// NETWORK 2
fbStation2(in_strUniqueId := 'Station 2', in_fbDevice := fbDevice2); // FB_ExampleStation
END_ACTION

ACTION A_Station3:
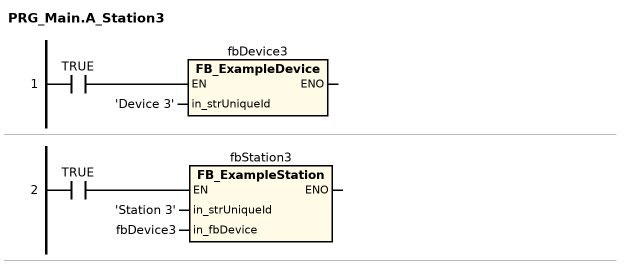
// NETWORK 1
fbDevice3(in_strUniqueId := 'Device 3'); // FB_ExampleDevice

// NETWORK 2
fbStation3(in_strUniqueId := 'Station 3', in_fbDevice := fbDevice3); // FB_ExampleStation
END_ACTION

ACTION A_Station4:
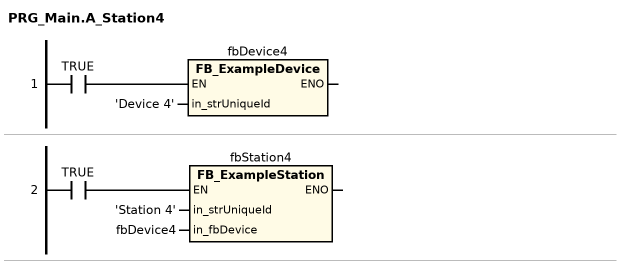
// NETWORK 1
fbDevice4(in_strUniqueId := 'Device 4'); // FB_ExampleDevice

// NETWORK 2
fbStation4(in_strUniqueId := 'Station 4', in_fbDevice := fbDevice4); // FB_ExampleStation
END_ACTION

METHOD M_TestCohapLibrary : BOOL

VAR
//	//Testing Cohap Related Vars

//	//Initialize Only	
//	MyCohapTest : FB_COHAP;
//	bInitializeCohapSystem: BOOL;
//	bRes_CohapConnected: BOOL;

//	//Execute RunImpMethods Only	;
//	bExecuteRunImpMethods: BOOL;
//	bRes_RunImpMethods: BOOL;

//	//Set Current Device Instance
//	bSetCurrentDevice_Cohap : BOOL;
//	bRes_SetCurrentDevice : BOOL;
//	//Input Params
//	strDeviceName : STRING;
	
//	//RunCommand
//	bRunCommandCohapSystem : BOOL;
//	bRes_RunCommand : BOOL;
//	//Input Params
//	strMethodName : STRING;
//	RunCom_InpuParams : T_CohapParameterList;
//	RunCom_ExpOutParamList : ARRAY[0..9] OF ST_ReturnParamsInfo;
//	//Output Params
//	RunCom_OutputParams : T_CohapParameterList;
	
//	//DummyTest Dictionary Prep for RunCommand Execution
//	RC_DT_InpPar : T_CohapParameterList;
//	RC_DT_ExpOutPL : ARRAY[0..9] OF ST_ReturnParamsInfo;
	
//	CohapMethodStrings : TMethodNames_Cohap;
//	CohapMethodControls : TMethod_Controls;
////	fbCohapHandler1: FB_COHAP;

/////////////////////////////////

//	// For readSerialNumber
//	readSerialNumber_inpuparams : T_CohapParameterList;
//	readSerialNumber_expoutparamlist : ARRAY[0..9] OF ST_ReturnParamsInfo;
//	readSerialNumber_outputparams : T_CohapParameterList;
	
//	// For ReadDeviceOutput
//	ReadDeviceOutput_inpuparams : T_CohapParameterList;
//	ReadDeviceOutput_expoutparamlist : ARRAY[0..9] OF ST_ReturnParamsInfo;
//	ReadDeviceOutput_outputparams : T_CohapParameterList;

	
//	// For PowerUp
//	PowerUp_inpuparams : T_CohapParameterList;
//	PowerUp_expoutparamlist : ARRAY[0..9] OF ST_ReturnParamsInfo;
//	PowerUp_outputparams : T_CohapParameterList;
	
//	// For PowerDown
//	PowerDown_inpuparams : T_CohapParameterList;
//	PowerDown_expoutparamlist : ARRAY[0..9] OF ST_ReturnParamsInfo;
//	PowerDown_outputparams : T_CohapParameterList;
	
//	// For TestDummy
//	TestDummy_inpuparams : T_CohapParameterList;
//	TestDummy_expoutparamlist : ARRAY[0..9] OF ST_ReturnParamsInfo;
//	TestDummy_outputparams : T_CohapParameterList;
	
//	// For TestDummy2
//	TestDummy2_inpuparams : T_CohapParameterList;
//	TestDummy2_expoutparamlist : ARRAY[0..9] OF ST_ReturnParamsInfo;
//	TestDummy2_outputparams : T_CohapParameterList;
	
//	// For init
//	init_inpuparams : T_CohapParameterList;
//	init_expoutparamlist : ARRAY[0..9] OF ST_ReturnParamsInfo;
//	init_outputparams : T_CohapParameterList;
	
//	// For getSICAndChannelCardVersions
//	getSICAndChannelCardVersions_inpuparams : T_CohapParameterList;
//	getSICAndChannelCardVersions_expoutparamlist : ARRAY[0..9] OF ST_ReturnParamsInfo;
//	getSICAndChannelCardVersions_outputparams : T_CohapParameterList;
	
//	// For getDLLVersions
//	getDLLVersions_inpuparams : T_CohapParameterList;
//	getDLLVersions_expoutparamlist : ARRAY[0..9] OF ST_ReturnParamsInfo;
//	getDLLVersions_outputparams : T_CohapParameterList;
	
//	// For initDUT
//	initDUT_inpuparams : T_CohapParameterList;
//	initDUT_expoutparamlist : ARRAY[0..9] OF ST_ReturnParamsInfo;
//	initDUT_outputparams : T_CohapParameterList;
	
//	//For Fast Channel Data
//	readFastChannelData_inputparams : T_CohapParameterList;
//	readFastChannelData_expoutparamlist : ARRAY[0..9] OF ST_ReturnParamsInfo;
//	readFastChannelData_outputparams : T_CohapParameterList;

//	// For T1 Step 1 Calibration
//	t1Step1_inpuparams : T_CohapParameterList;
//	t1Step1_expoutparamlist : ARRAY[0..9] OF ST_ReturnParamsInfo;
//	t1Step1_outputparams : T_CohapParameterList;
	
////	// For T1 Step 2 Calibration
////	t1Step2_inpuparams : T_CohapParameterList;
////	t1Step2_expoutparamlist : ARRAY[0..9] OF ST_ReturnParamsInfo;
////	t1Step2_outputparams : T_CohapParameterList;
	
////	// For T1 Step 3 Calibration
////	t1Step3_inpuparams : T_CohapParameterList;
////	t1Step3_expoutparamlist : ARRAY[0..9] OF ST_ReturnParamsInfo;
////	t1Step3_outputparams : T_CohapParameterList;
	
//	// For T2 Step 1 Calibration
//	t2Step1_inpuparams : T_CohapParameterList;
//	t2Step1_expoutparamlist : ARRAY[0..9] OF ST_ReturnParamsInfo;
//	t2Step1_outputparams : T_CohapParameterList;
	
//	// For T2 Step 2 Calibration
//	t2Step2_inpuparams : T_CohapParameterList;
//	t2Step2_expoutparamlist : ARRAY[0..9] OF ST_ReturnParamsInfo;
//	t2Step2_outputparams : T_CohapParameterList;
	
//	// For T2 Step 3 Calibration
//	t2Step3_inpuparams : T_CohapParameterList;
//	t2Step3_expoutparamlist : ARRAY[0..9] OF ST_ReturnParamsInfo;
//	t2Step3_outputparams : T_CohapParameterList;
	
//	// InitLot Device12133 class in Mech Device Lib Calibration
//	InitLot_inputparams : T_CohapParameterList;
//	InitLot_expoutparamlist : ARRAY[0..9] OF ST_ReturnParamsInfo;
//	InitLot_outputparams : T_CohapParameterList;
	
////	//For Init Lot
////	InitLot_inputparams : T_CohapParameterList;
////	InitLot_expoutparamlist : ARRAY[0..9] OF ST_ReturnParamsInfo;
////	InitLot_outputparams : T_CohapParameterList;	
//	// For T1 Step 1 Calibration
//	t1Precal_inputparams : T_CohapParameterList;
//	t1Precal_expoutparamlist : ARRAY[0..9] OF ST_ReturnParamsInfo;
//	t1Precal_outputparams : T_CohapParameterList;
//	// For T1 Step 2 Calibration
//	t1Step2_inputparams : T_CohapParameterList;
//	t1Step2_expoutparamlist : ARRAY[0..9] OF ST_ReturnParamsInfo;
//	t1Step2_outputparams : T_CohapParameterList;
//	// For T1 Step 3 Calibration
//	t1Step3_inputparams : T_CohapParameterList;
//	t1Step3_expoutparamlist : ARRAY[0..9] OF ST_ReturnParamsInfo;
//	t1Step3_outputparams : T_CohapParameterList;
END_VAR
VAR_INST // added by the converter: edge detectors and wires of the graphical bodies
    _w1, _w2, _w3, _w4, _w5, _w6, _w7, _w8, _w9, _w10, _w11, _w12, _w13, _w14, _w15, _w16, _w17, _w18, _w19, _w20, _w21, _w22, _w23, _w24, _w25, _w26, _w27, _w28, _w29, _w30, _w31, _w32, _w33, _w34, _w35, _w36, _w37, _w38, _w39, _w40 : BOOL;
END_VAR
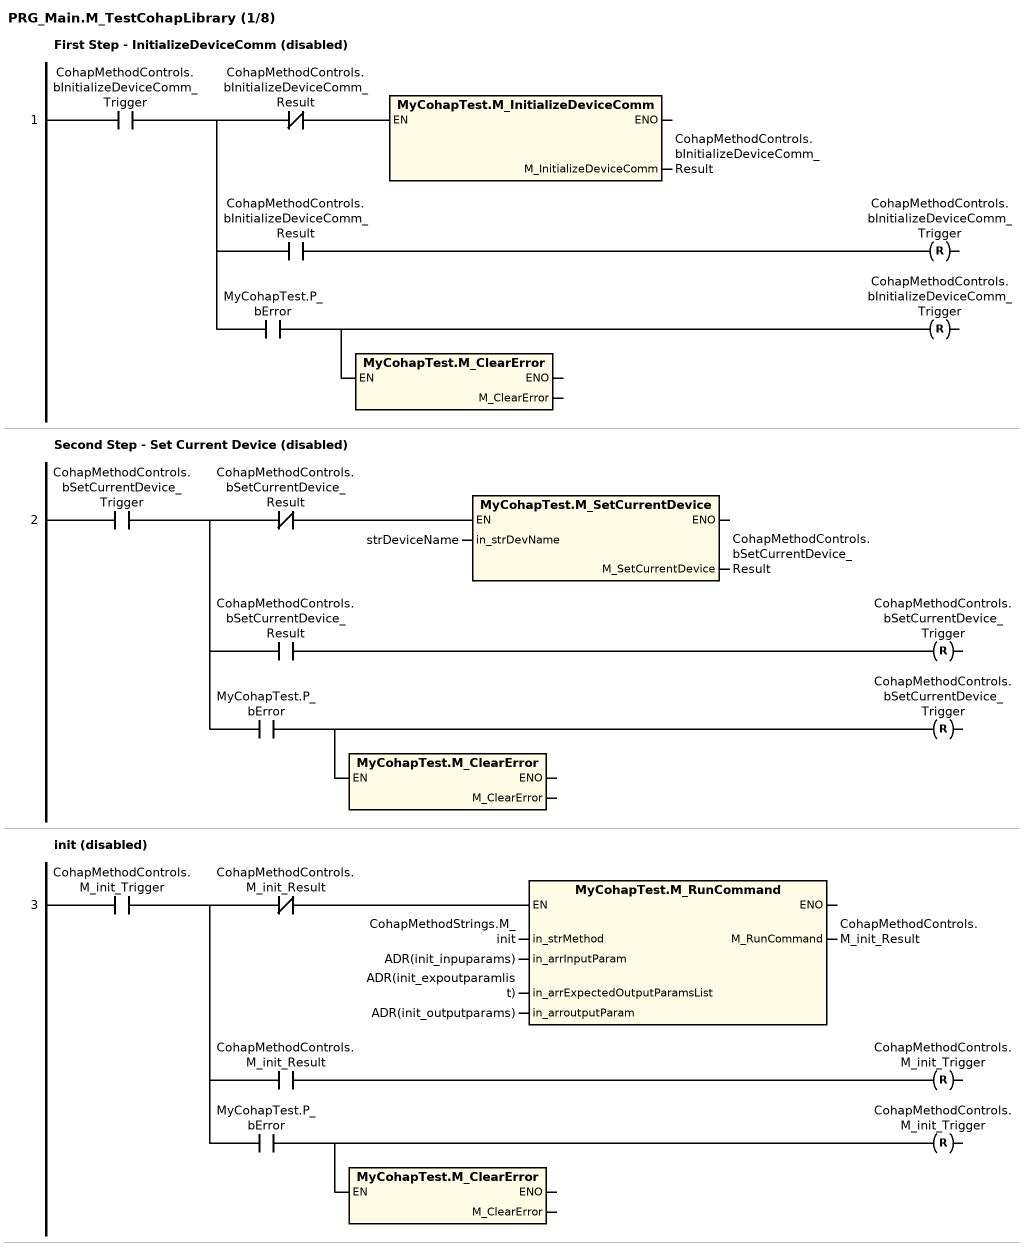
// NETWORK 1: First Step - InitializeDeviceComm (disabled)
// _w1 := CohapMethodControls.bInitializeDeviceComm_Trigger;
// IF _w1 AND NOT CohapMethodControls.bInitializeDeviceComm_Result THEN
//     CohapMethodControls.bInitializeDeviceComm_Result := MyCohapTest.M_InitializeDeviceComm();
// END_IF
// CohapMethodControls.bInitializeDeviceComm_Trigger R= _w1 AND CohapMethodControls.bInitializeDeviceComm_Result;
// _w2 := _w1 AND MyCohapTest.P_bError;
// CohapMethodControls.bInitializeDeviceComm_Trigger R= _w2;
// IF _w2 THEN MyCohapTest.M_ClearError(); END_IF

// NETWORK 2: Second Step - Set Current Device (disabled)
// _w3 := CohapMethodControls.bSetCurrentDevice_Trigger;
// IF _w3 AND NOT CohapMethodControls.bSetCurrentDevice_Result THEN
//     CohapMethodControls.bSetCurrentDevice_Result := MyCohapTest.M_SetCurrentDevice(in_strDevName := strDeviceName);
// END_IF
// CohapMethodControls.bSetCurrentDevice_Trigger R= _w3 AND CohapMethodControls.bSetCurrentDevice_Result;
// _w4 := _w3 AND MyCohapTest.P_bError;
// CohapMethodControls.bSetCurrentDevice_Trigger R= _w4;
// IF _w4 THEN MyCohapTest.M_ClearError(); END_IF

// NETWORK 3: init (disabled)
// _w5 := CohapMethodControls.M_init_Trigger;
// IF _w5 AND NOT CohapMethodControls.M_init_Result THEN
//     CohapMethodControls.M_init_Result := MyCohapTest.M_RunCommand(in_strMethod := CohapMethodStrings.M_init, in_arrInputParam := ADR(init_inpuparams), in_arrExpectedOutputParamsList := ADR(init_expoutparamlist), in_arroutputParam := ADR(init_outputparams));
// END_IF
// CohapMethodControls.M_init_Trigger R= _w5 AND CohapMethodControls.M_init_Result;
// _w6 := _w5 AND MyCohapTest.P_bError;
// CohapMethodControls.M_init_Trigger R= _w6;
// IF _w6 THEN MyCohapTest.M_ClearError(); END_IF

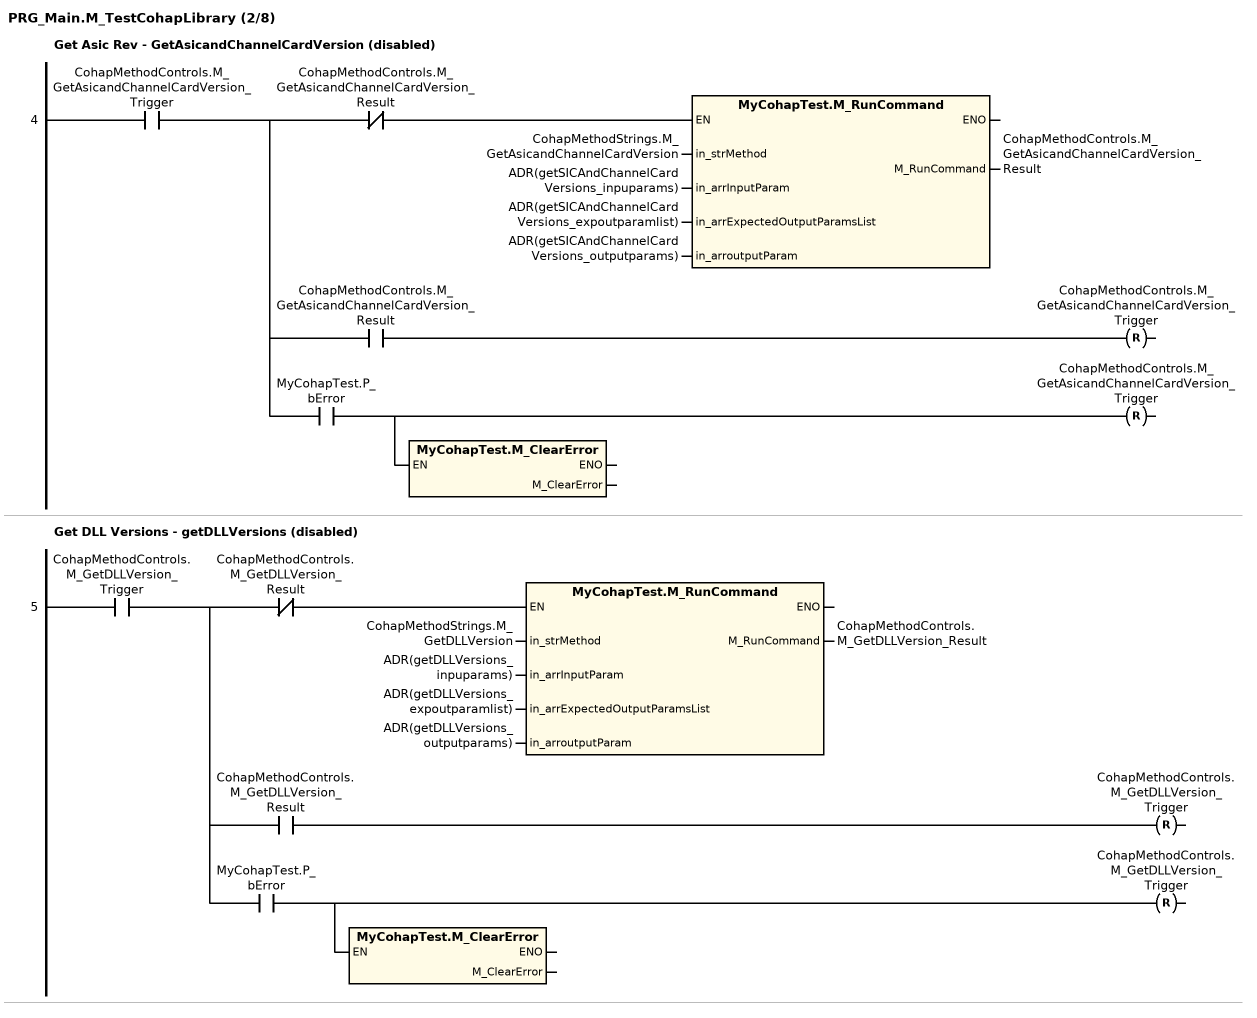
// NETWORK 4: Get Asic Rev - GetAsicandChannelCardVersion (disabled)
// _w7 := CohapMethodControls.M_GetAsicandChannelCardVersion_Trigger;
// IF _w7 AND NOT CohapMethodControls.M_GetAsicandChannelCardVersion_Result THEN
//     CohapMethodControls.M_GetAsicandChannelCardVersion_Result := MyCohapTest.M_RunCommand(in_strMethod := CohapMethodStrings.M_GetAsicandChannelCardVersion, in_arrInputParam := ADR(getSICAndChannelCardVersions_inpuparams), in_arrExpectedOutputParamsList := ADR(getSICAndChannelCardVersions_expoutparamlist), in_arroutputParam := ADR(getSICAndChannelCardVersions_outputparams));
// END_IF
// CohapMethodControls.M_GetAsicandChannelCardVersion_Trigger R= _w7 AND CohapMethodControls.M_GetAsicandChannelCardVersion_Result;
// _w8 := _w7 AND MyCohapTest.P_bError;
// CohapMethodControls.M_GetAsicandChannelCardVersion_Trigger R= _w8;
// IF _w8 THEN MyCohapTest.M_ClearError(); END_IF

// NETWORK 5: Get DLL Versions - getDLLVersions (disabled)
// _w9 := CohapMethodControls.M_GetDLLVersion_Trigger;
// IF _w9 AND NOT CohapMethodControls.M_GetDLLVersion_Result THEN
//     CohapMethodControls.M_GetDLLVersion_Result := MyCohapTest.M_RunCommand(in_strMethod := CohapMethodStrings.M_GetDLLVersion, in_arrInputParam := ADR(getDLLVersions_inpuparams), in_arrExpectedOutputParamsList := ADR(getDLLVersions_expoutparamlist), in_arroutputParam := ADR(getDLLVersions_outputparams));
// END_IF
// CohapMethodControls.M_GetDLLVersion_Trigger R= _w9 AND CohapMethodControls.M_GetDLLVersion_Result;
// _w10 := _w9 AND MyCohapTest.P_bError;
// CohapMethodControls.M_GetDLLVersion_Trigger R= _w10;
// IF _w10 THEN MyCohapTest.M_ClearError(); END_IF

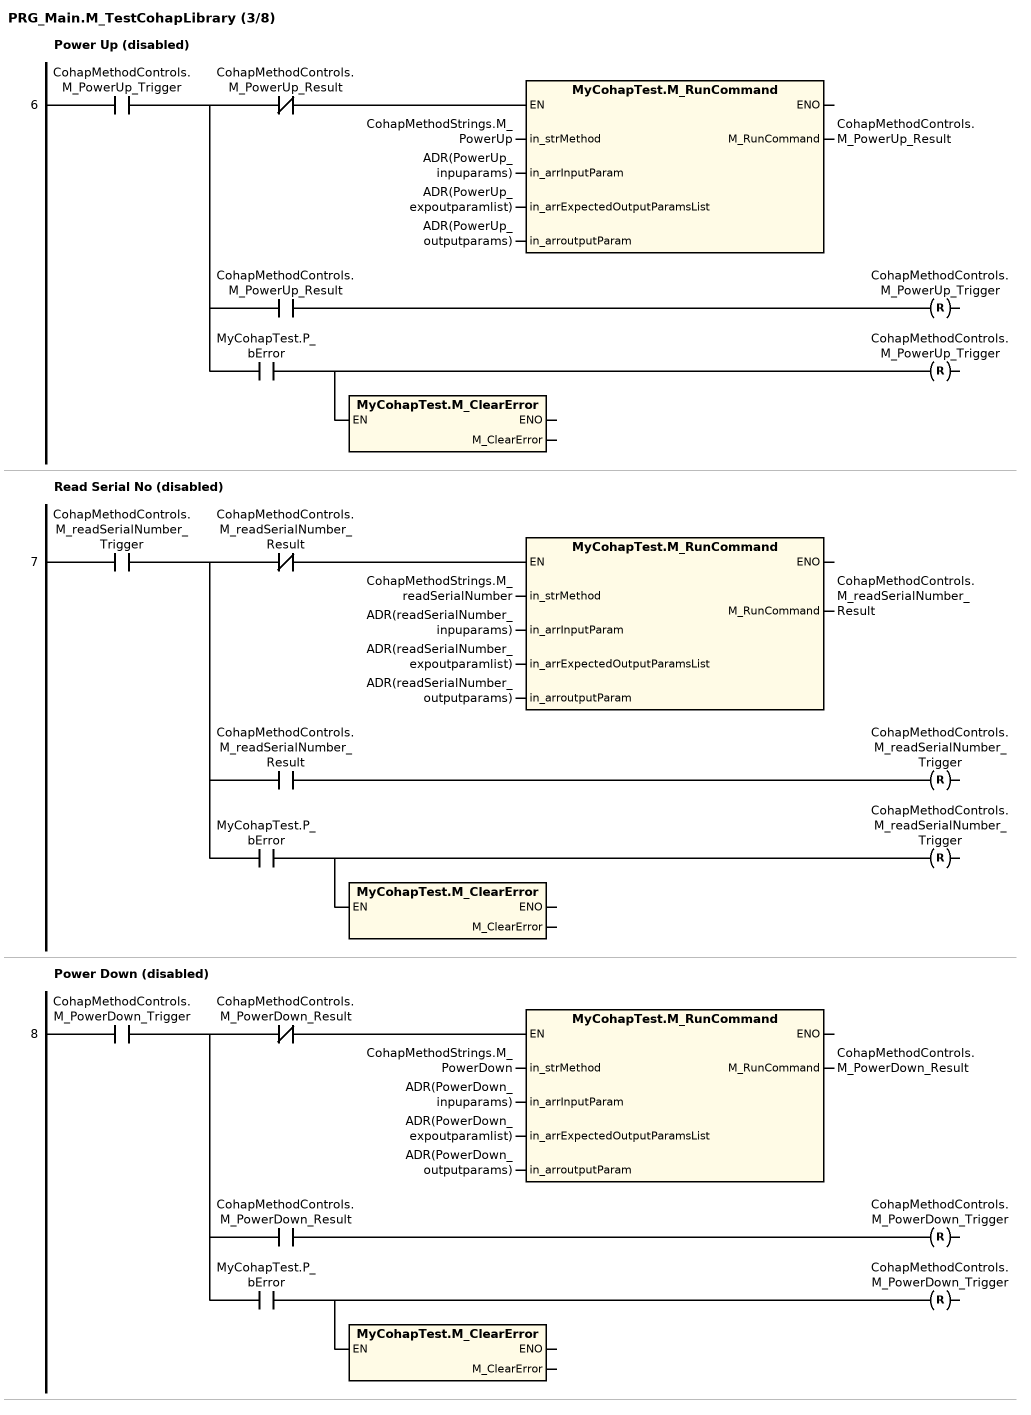
// NETWORK 6: Power Up (disabled)
// _w11 := CohapMethodControls.M_PowerUp_Trigger;
// IF _w11 AND NOT CohapMethodControls.M_PowerUp_Result THEN
//     CohapMethodControls.M_PowerUp_Result := MyCohapTest.M_RunCommand(in_strMethod := CohapMethodStrings.M_PowerUp, in_arrInputParam := ADR(PowerUp_inpuparams), in_arrExpectedOutputParamsList := ADR(PowerUp_expoutparamlist), in_arroutputParam := ADR(PowerUp_outputparams));
// END_IF
// CohapMethodControls.M_PowerUp_Trigger R= _w11 AND CohapMethodControls.M_PowerUp_Result;
// _w12 := _w11 AND MyCohapTest.P_bError;
// CohapMethodControls.M_PowerUp_Trigger R= _w12;
// IF _w12 THEN MyCohapTest.M_ClearError(); END_IF

// NETWORK 7: Read Serial No (disabled)
// _w13 := CohapMethodControls.M_readSerialNumber_Trigger;
// IF _w13 AND NOT CohapMethodControls.M_readSerialNumber_Result THEN
//     CohapMethodControls.M_readSerialNumber_Result := MyCohapTest.M_RunCommand(in_strMethod := CohapMethodStrings.M_readSerialNumber, in_arrInputParam := ADR(readSerialNumber_inpuparams), in_arrExpectedOutputParamsList := ADR(readSerialNumber_expoutparamlist), in_arroutputParam := ADR(readSerialNumber_outputparams));
// END_IF
// CohapMethodControls.M_readSerialNumber_Trigger R= _w13 AND CohapMethodControls.M_readSerialNumber_Result;
// _w14 := _w13 AND MyCohapTest.P_bError;
// CohapMethodControls.M_readSerialNumber_Trigger R= _w14;
// IF _w14 THEN MyCohapTest.M_ClearError(); END_IF

// NETWORK 8: Power Down (disabled)
// _w15 := CohapMethodControls.M_PowerDown_Trigger;
// IF _w15 AND NOT CohapMethodControls.M_PowerDown_Result THEN
//     CohapMethodControls.M_PowerDown_Result := MyCohapTest.M_RunCommand(in_strMethod := CohapMethodStrings.M_PowerDown, in_arrInputParam := ADR(PowerDown_inpuparams), in_arrExpectedOutputParamsList := ADR(PowerDown_expoutparamlist), in_arroutputParam := ADR(PowerDown_outputparams));
// END_IF
// CohapMethodControls.M_PowerDown_Trigger R= _w15 AND CohapMethodControls.M_PowerDown_Result;
// _w16 := _w15 AND MyCohapTest.P_bError;
// CohapMethodControls.M_PowerDown_Trigger R= _w16;
// IF _w16 THEN MyCohapTest.M_ClearError(); END_IF

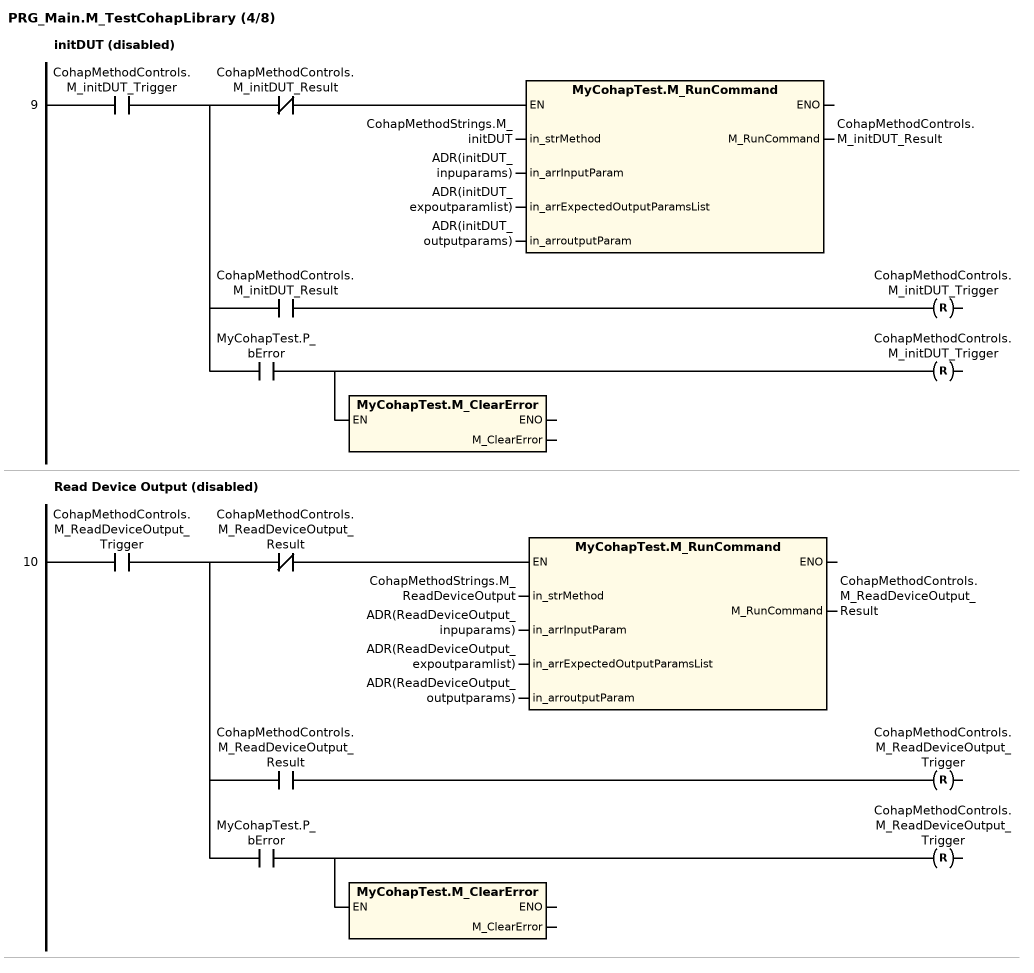
// NETWORK 9: initDUT (disabled)
// _w17 := CohapMethodControls.M_initDUT_Trigger;
// IF _w17 AND NOT CohapMethodControls.M_initDUT_Result THEN
//     CohapMethodControls.M_initDUT_Result := MyCohapTest.M_RunCommand(in_strMethod := CohapMethodStrings.M_initDUT, in_arrInputParam := ADR(initDUT_inpuparams), in_arrExpectedOutputParamsList := ADR(initDUT_expoutparamlist), in_arroutputParam := ADR(initDUT_outputparams));
// END_IF
// CohapMethodControls.M_initDUT_Trigger R= _w17 AND CohapMethodControls.M_initDUT_Result;
// _w18 := _w17 AND MyCohapTest.P_bError;
// CohapMethodControls.M_initDUT_Trigger R= _w18;
// IF _w18 THEN MyCohapTest.M_ClearError(); END_IF

// NETWORK 10: Read Device Output (disabled)
// _w19 := CohapMethodControls.M_ReadDeviceOutput_Trigger;
// IF _w19 AND NOT CohapMethodControls.M_ReadDeviceOutput_Result THEN
//     CohapMethodControls.M_ReadDeviceOutput_Result := MyCohapTest.M_RunCommand(in_strMethod := CohapMethodStrings.M_ReadDeviceOutput, in_arrInputParam := ADR(ReadDeviceOutput_inpuparams), in_arrExpectedOutputParamsList := ADR(ReadDeviceOutput_expoutparamlist), in_arroutputParam := ADR(ReadDeviceOutput_outputparams));
// END_IF
// CohapMethodControls.M_ReadDeviceOutput_Trigger R= _w19 AND CohapMethodControls.M_ReadDeviceOutput_Result;
// _w20 := _w19 AND MyCohapTest.P_bError;
// CohapMethodControls.M_ReadDeviceOutput_Trigger R= _w20;
// IF _w20 THEN MyCohapTest.M_ClearError(); END_IF

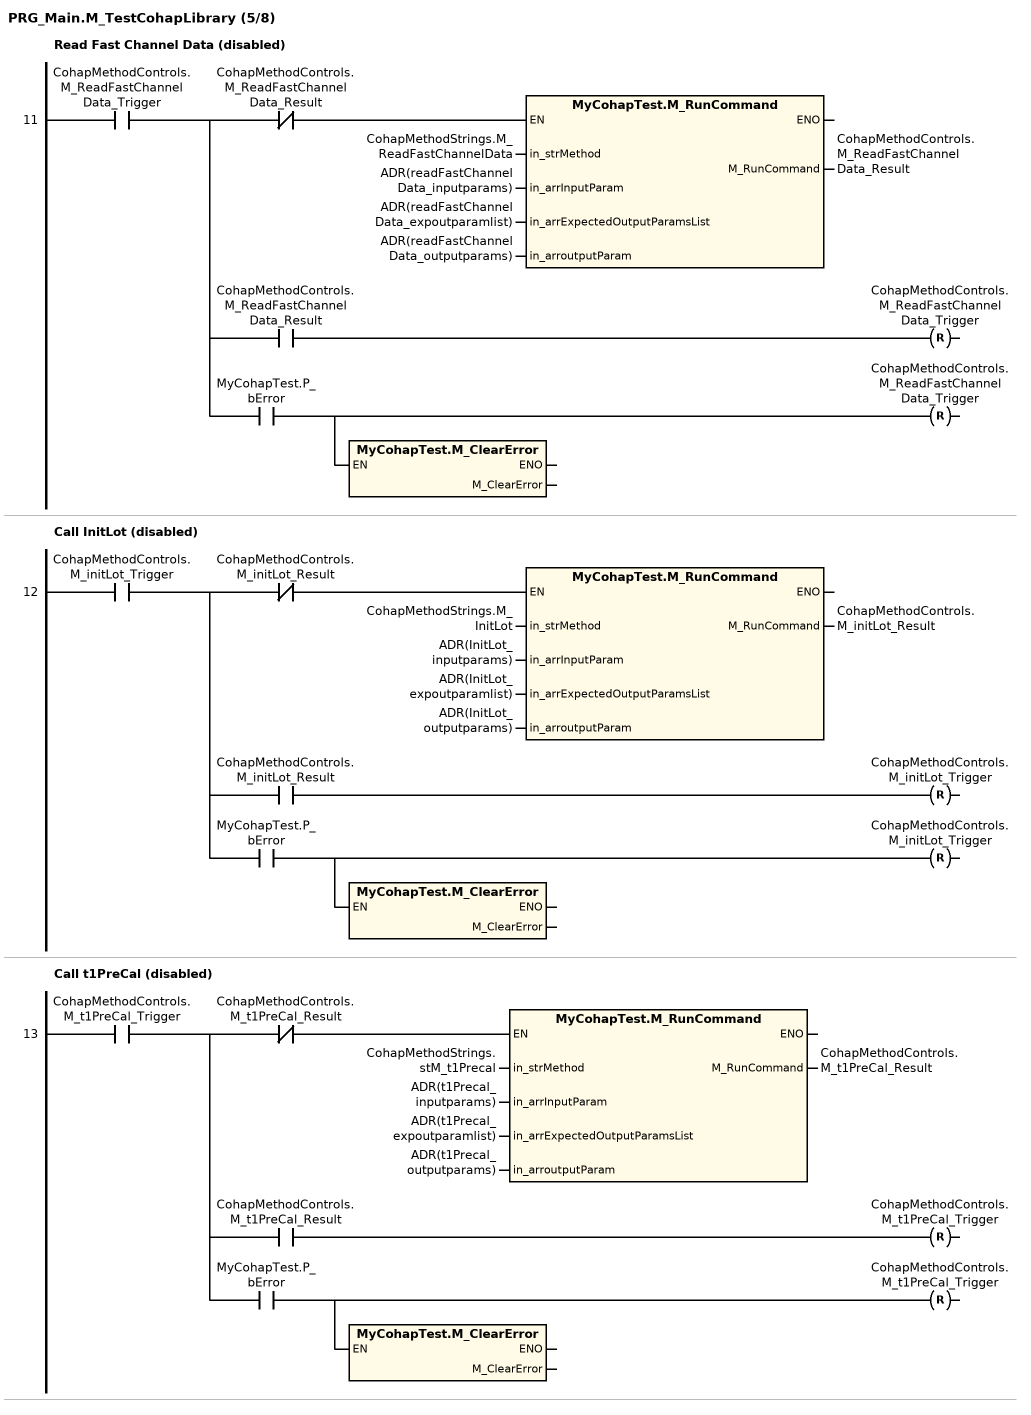
// NETWORK 11: Read Fast Channel Data (disabled)
// _w21 := CohapMethodControls.M_ReadFastChannelData_Trigger;
// IF _w21 AND NOT CohapMethodControls.M_ReadFastChannelData_Result THEN
//     CohapMethodControls.M_ReadFastChannelData_Result := MyCohapTest.M_RunCommand(in_strMethod := CohapMethodStrings.M_ReadFastChannelData, in_arrInputParam := ADR(readFastChannelData_inputparams), in_arrExpectedOutputParamsList := ADR(readFastChannelData_expoutparamlist), in_arroutputParam := ADR(readFastChannelData_outputparams));
// END_IF
// CohapMethodControls.M_ReadFastChannelData_Trigger R= _w21 AND CohapMethodControls.M_ReadFastChannelData_Result;
// _w22 := _w21 AND MyCohapTest.P_bError;
// CohapMethodControls.M_ReadFastChannelData_Trigger R= _w22;
// IF _w22 THEN MyCohapTest.M_ClearError(); END_IF

// NETWORK 12: Call InitLot (disabled)
// _w23 := CohapMethodControls.M_initLot_Trigger;
// IF _w23 AND NOT CohapMethodControls.M_initLot_Result THEN
//     CohapMethodControls.M_initLot_Result := MyCohapTest.M_RunCommand(in_strMethod := CohapMethodStrings.M_InitLot, in_arrInputParam := ADR(InitLot_inputparams), in_arrExpectedOutputParamsList := ADR(InitLot_expoutparamlist), in_arroutputParam := ADR(InitLot_outputparams));
// END_IF
// CohapMethodControls.M_initLot_Trigger R= _w23 AND CohapMethodControls.M_initLot_Result;
// _w24 := _w23 AND MyCohapTest.P_bError;
// CohapMethodControls.M_initLot_Trigger R= _w24;
// IF _w24 THEN MyCohapTest.M_ClearError(); END_IF

// NETWORK 13: Call t1PreCal (disabled)
// _w25 := CohapMethodControls.M_t1PreCal_Trigger;
// IF _w25 AND NOT CohapMethodControls.M_t1PreCal_Result THEN
//     CohapMethodControls.M_t1PreCal_Result := MyCohapTest.M_RunCommand(in_strMethod := CohapMethodStrings.stM_t1Precal, in_arrInputParam := ADR(t1Precal_inputparams), in_arrExpectedOutputParamsList := ADR(t1Precal_expoutparamlist), in_arroutputParam := ADR(t1Precal_outputparams));
// END_IF
// CohapMethodControls.M_t1PreCal_Trigger R= _w25 AND CohapMethodControls.M_t1PreCal_Result;
// _w26 := _w25 AND MyCohapTest.P_bError;
// CohapMethodControls.M_t1PreCal_Trigger R= _w26;
// IF _w26 THEN MyCohapTest.M_ClearError(); END_IF

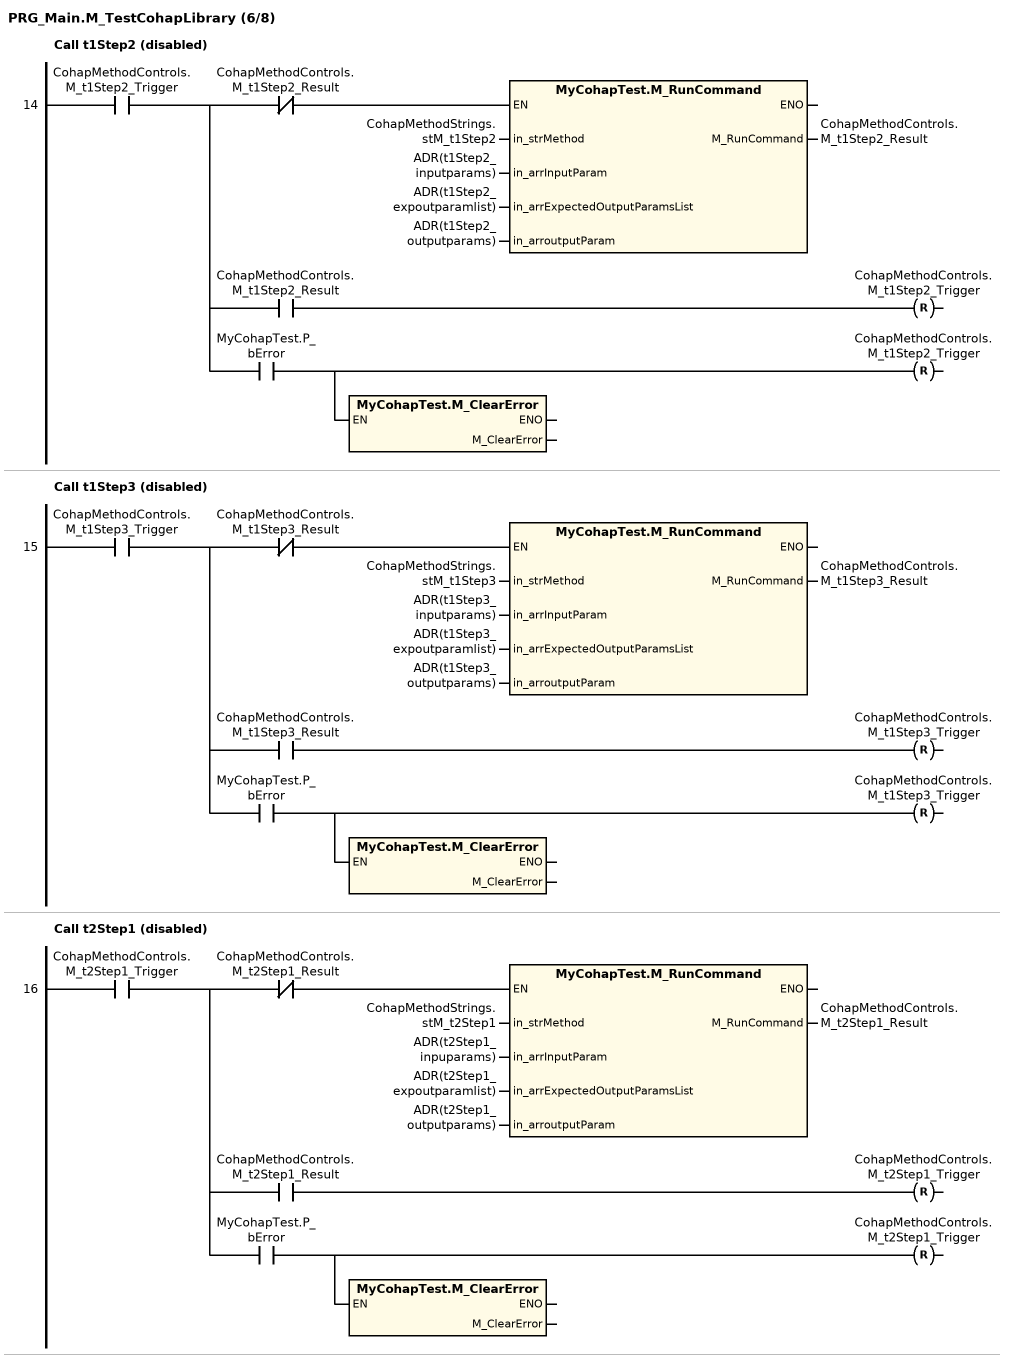
// NETWORK 14: Call t1Step2 (disabled)
// _w27 := CohapMethodControls.M_t1Step2_Trigger;
// IF _w27 AND NOT CohapMethodControls.M_t1Step2_Result THEN
//     CohapMethodControls.M_t1Step2_Result := MyCohapTest.M_RunCommand(in_strMethod := CohapMethodStrings.stM_t1Step2, in_arrInputParam := ADR(t1Step2_inputparams), in_arrExpectedOutputParamsList := ADR(t1Step2_expoutparamlist), in_arroutputParam := ADR(t1Step2_outputparams));
// END_IF
// CohapMethodControls.M_t1Step2_Trigger R= _w27 AND CohapMethodControls.M_t1Step2_Result;
// _w28 := _w27 AND MyCohapTest.P_bError;
// CohapMethodControls.M_t1Step2_Trigger R= _w28;
// IF _w28 THEN MyCohapTest.M_ClearError(); END_IF

// NETWORK 15: Call t1Step3 (disabled)
// _w29 := CohapMethodControls.M_t1Step3_Trigger;
// IF _w29 AND NOT CohapMethodControls.M_t1Step3_Result THEN
//     CohapMethodControls.M_t1Step3_Result := MyCohapTest.M_RunCommand(in_strMethod := CohapMethodStrings.stM_t1Step3, in_arrInputParam := ADR(t1Step3_inputparams), in_arrExpectedOutputParamsList := ADR(t1Step3_expoutparamlist), in_arroutputParam := ADR(t1Step3_outputparams));
// END_IF
// CohapMethodControls.M_t1Step3_Trigger R= _w29 AND CohapMethodControls.M_t1Step3_Result;
// _w30 := _w29 AND MyCohapTest.P_bError;
// CohapMethodControls.M_t1Step3_Trigger R= _w30;
// IF _w30 THEN MyCohapTest.M_ClearError(); END_IF

// NETWORK 16: Call t2Step1 (disabled)
// _w31 := CohapMethodControls.M_t2Step1_Trigger;
// IF _w31 AND NOT CohapMethodControls.M_t2Step1_Result THEN
//     CohapMethodControls.M_t2Step1_Result := MyCohapTest.M_RunCommand(in_strMethod := CohapMethodStrings.stM_t2Step1, in_arrInputParam := ADR(t2Step1_inpuparams), in_arrExpectedOutputParamsList := ADR(t2Step1_expoutparamlist), in_arroutputParam := ADR(t2Step1_outputparams));
// END_IF
// CohapMethodControls.M_t2Step1_Trigger R= _w31 AND CohapMethodControls.M_t2Step1_Result;
// _w32 := _w31 AND MyCohapTest.P_bError;
// CohapMethodControls.M_t2Step1_Trigger R= _w32;
// IF _w32 THEN MyCohapTest.M_ClearError(); END_IF

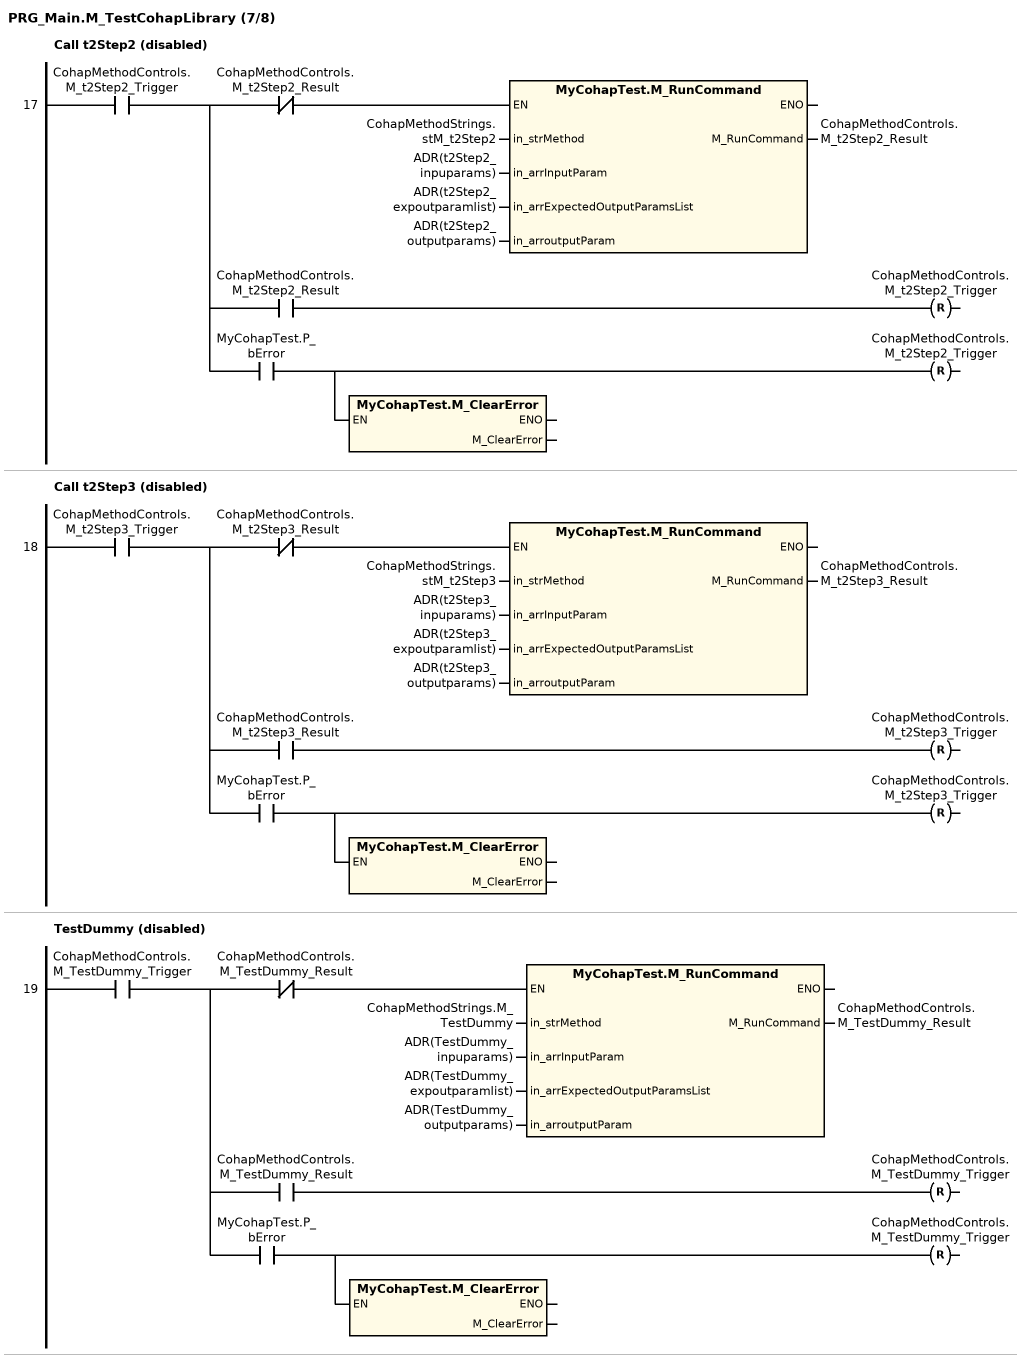
// NETWORK 17: Call t2Step2 (disabled)
// _w33 := CohapMethodControls.M_t2Step2_Trigger;
// IF _w33 AND NOT CohapMethodControls.M_t2Step2_Result THEN
//     CohapMethodControls.M_t2Step2_Result := MyCohapTest.M_RunCommand(in_strMethod := CohapMethodStrings.stM_t2Step2, in_arrInputParam := ADR(t2Step2_inpuparams), in_arrExpectedOutputParamsList := ADR(t2Step2_expoutparamlist), in_arroutputParam := ADR(t2Step2_outputparams));
// END_IF
// CohapMethodControls.M_t2Step2_Trigger R= _w33 AND CohapMethodControls.M_t2Step2_Result;
// _w34 := _w33 AND MyCohapTest.P_bError;
// CohapMethodControls.M_t2Step2_Trigger R= _w34;
// IF _w34 THEN MyCohapTest.M_ClearError(); END_IF

// NETWORK 18: Call t2Step3 (disabled)
// _w35 := CohapMethodControls.M_t2Step3_Trigger;
// IF _w35 AND NOT CohapMethodControls.M_t2Step3_Result THEN
//     CohapMethodControls.M_t2Step3_Result := MyCohapTest.M_RunCommand(in_strMethod := CohapMethodStrings.stM_t2Step3, in_arrInputParam := ADR(t2Step3_inpuparams), in_arrExpectedOutputParamsList := ADR(t2Step3_expoutparamlist), in_arroutputParam := ADR(t2Step3_outputparams));
// END_IF
// CohapMethodControls.M_t2Step3_Trigger R= _w35 AND CohapMethodControls.M_t2Step3_Result;
// _w36 := _w35 AND MyCohapTest.P_bError;
// CohapMethodControls.M_t2Step3_Trigger R= _w36;
// IF _w36 THEN MyCohapTest.M_ClearError(); END_IF

// NETWORK 19: TestDummy (disabled)
// _w37 := CohapMethodControls.M_TestDummy_Trigger;
// IF _w37 AND NOT CohapMethodControls.M_TestDummy_Result THEN
//     CohapMethodControls.M_TestDummy_Result := MyCohapTest.M_RunCommand(in_strMethod := CohapMethodStrings.M_TestDummy, in_arrInputParam := ADR(TestDummy_inpuparams), in_arrExpectedOutputParamsList := ADR(TestDummy_expoutparamlist), in_arroutputParam := ADR(TestDummy_outputparams));
// END_IF
// CohapMethodControls.M_TestDummy_Trigger R= _w37 AND CohapMethodControls.M_TestDummy_Result;
// _w38 := _w37 AND MyCohapTest.P_bError;
// CohapMethodControls.M_TestDummy_Trigger R= _w38;
// IF _w38 THEN MyCohapTest.M_ClearError(); END_IF

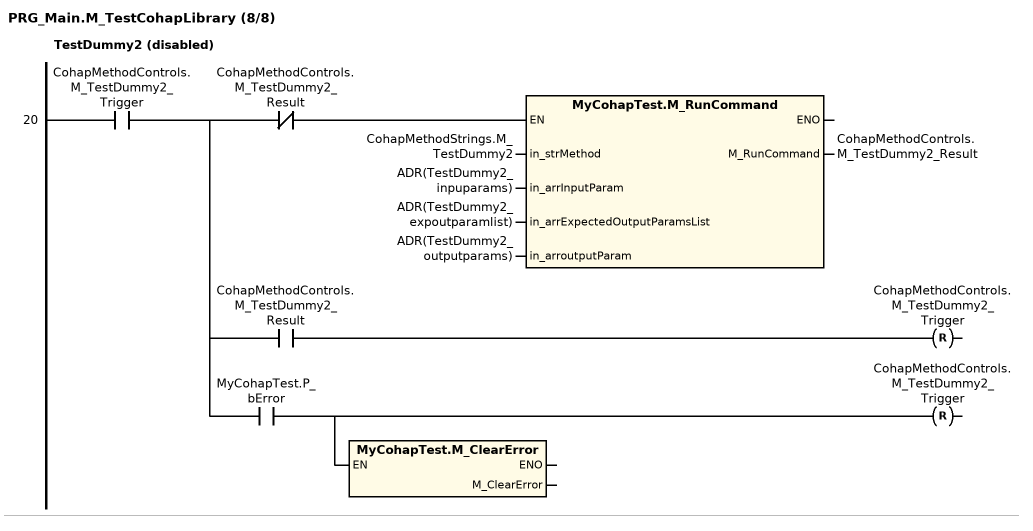
// NETWORK 20: TestDummy2 (disabled)
// _w39 := CohapMethodControls.M_TestDummy2_Trigger;
// IF _w39 AND NOT CohapMethodControls.M_TestDummy2_Result THEN
//     CohapMethodControls.M_TestDummy2_Result := MyCohapTest.M_RunCommand(in_strMethod := CohapMethodStrings.M_TestDummy2, in_arrInputParam := ADR(TestDummy2_inpuparams), in_arrExpectedOutputParamsList := ADR(TestDummy2_expoutparamlist), in_arroutputParam := ADR(TestDummy2_outputparams));
// END_IF
// CohapMethodControls.M_TestDummy2_Trigger R= _w39 AND CohapMethodControls.M_TestDummy2_Result;
// _w40 := _w39 AND MyCohapTest.P_bError;
// CohapMethodControls.M_TestDummy2_Trigger R= _w40;
// IF _w40 THEN MyCohapTest.M_ClearError(); END_IF
END_METHOD

METHOD M_TestLaserMarker : BOOL
VAR_INPUT
END_VAR
VAR
		bConnectToLaserMarker: BOOL;
	bRes_LaserConnected: BOOL;
	bTestADSServer: BOOL;
	strTarget: T_MaxString;
	strCommand: T_MaxString;
	arrParams: T_ApiMethodParameters;
	MyResults: T_MaxString;
	bInterfaceTest : BOOL;
	temp: BOOL;
	bDisconnectFromLaserMarker: BOOL;
	bRes_LaserDisconnected: BOOL;
	bPeakCurrentProgramInLaser: BOOL;
	bRes_PeakCurrentProgramInLaser: BOOL;
	bSendProgramToLaser: BOOL;
	bRes_SendProgramtoLaser: BOOL;
	filepath : STRING;
	LaserMemoryLocation : INT;
	bSaveCurrentLaserProgramtoPC : BOOL;
	bRes_SaveCurrentLaserProgramtoPC: BOOL;
	LaserProgramFolderPath: STRING;
	bGetCurrentProgram : BOOL;
	bRes_GetCurrentProgram : BOOL;
	CurrentProgramName : T_MaxString;
	bStartMarking: BOOL;
	bRes_StartMarking: BOOL;
	bStopMarking: BOOL;
	bRes_StopMarking: BOOL;
	bClearLaserErrors: BOOL;
	bRes_ClearLaserErrors: BOOL;
	bUpdateProgramBlockInTheLaser: BOOL;
	bRes_UpdateProgramBlockInTheLaser: BOOL;
	_blockNumber: INT;
	_blockData: STRING;
	_blockType : BlockTypes;
	bGetLaserStatus: BOOL;
	bRes_GetLaserStatus: BOOL;
	_string_laserstatus : STRING;
	bGetLaserErrorStatus: BOOL;
	bRes_GetLaserErrorStatus: BOOL;
	_bIsLaserError : BOOL;
	bGetLaserActivatedStatus: BOOL;
	bRes_GetLaserActivatedStatus: BOOL;
	_bIsLaserActivated : BOOL;
	bGetLaserMarkingStatus: BOOL;
	bRes_GetLaserMarkingStatus: BOOL;
	_bIsLaserMarking : BOOL;
	bRes_Reset: BOOL;
	bResetErrors: BOOL;
	bUpdateProgramBlockMarkEnabledInTheLaser: BOOL;
	bRes_UpdateProgramBlockMarkEnabledInTheLaser: BOOL;
	_bool_markenabled : BOOL;
	_blockType_enum : BlockTypes;
	UpdateSingleBlockMarkEnabledIntheLaser_Success: BOOL;
	_bUpdateSingleBlockDataSuccess : BOOL;
	_bUpdateSingleBlockMarkEnabled_Success : BOOL;
	bUpdateAllMarkingInfo: BOOL;
	LastBlockToMark : INT;
	_OneTimeArrayBuild : BOOL := TRUE;
	BlockInfoArray : ARRAY [0..255] OF OneBlockInfo;
	bRes_UpdateAllMarkingInfo: BOOL;
	intIndex: INT;
	intIndex2 : INT;
	inst_intStep: INT := 0;
	_tempString : STRING;
	bRes_UpdateAllMarkInfo : ARRAY [0..255] OF BOOL;
	bUpdateAllMarkingInfo_MethodCall: BOOL;
	bRes_UpdateAllMarkingInfo_MethodCall: BOOL;
	fbDataHandler: FB_DataTracker;
	fbDataHandler2: FB_DataTracker;
	fbDatabaseCommandRouter: FB_AdsCommandRouter;
	_inst_bDataTransferred: BOOL;
	// (* Name of the parameters database transfer ID. *)
	in_strParametersDatabaseName: T_MaxString := 'GetLimits';
	in_strParametersDBNameLaserLimits_L1 : T_MaxString := 'GetLaserMarkingParams_L1';
	in_strParametersDBNameLaserLimits_L2 : T_MaxString := 'GetLaserMarkingParams_L2';
	in_strParametersDBNameLaserLimits_R1 : T_MaxString := 'GetLaserMarkingParams_R1';
	in_strParametersDBNameLaserLimits_R2 : T_MaxString := 'GetLaserMarkingParams_R2';	
	_inst_bLaserLimitsDataTransferred_L1 : BOOL;
	_inst_bLaserLimitsDataTransferred_L2 : BOOL;
	_inst_bLaserLimitsDataTransferred_R1 : BOOL;
	_inst_bLaserLimitsDataTransferred_R2 : BOOL;
	bGetLimitsFromDB : BOOL;
	bGetLaserParamsFromDB_L1 : BOOL;
	bGetLaserParamsFromDB_L2 : BOOL;
	bGetLaserParamsFromDB_R1 : BOOL;
	bGetLaserParamsFromDB_R2 : BOOL;
	bPerformPriorOp_Smart: BOOL;
	in_strParametersDBName_SmartWater : T_MaxString := 'GetPriorOPA';
	_inst_bPriorOp_Smart: BOOL;
	
	bPerformPriorOp_FFT: BOOL;
	in_strParametersDBName_FFTLaser_L1 : T_MaxString := 'LaserMarkCheckL1';
	_inst_bPriorOp_FFT: BOOL;
	
	Temp_CR_LOOKUP_NestL1 : INT;
	iLengthDataMatrixNestL1 : INT;
	ParamsArrayNestA : STRING;
END_VAR
//IF bConnectToLaserMarker THEN
//	bRes_LaserConnected := MyLaser1.M_Connect();
//	IF bRes_LaserConnected THEN
//	//Add some timer based logic to do error handling.
//		bConnectToLaserMarker := FALSE;
//	ELSIF MyLaser1.P_bError THEN
//		bConnectToLaserMarker := FALSE;
//		MyLaser1.M_ClearError();
//	END_IF
//END_IF


//IF bDisconnectFromLaserMarker THEN
//	bRes_LaserDisconnected := MyLaser1.M_Disconnect();
//	IF bRes_LaserDisconnected THEN
//		bDisconnectFromLaserMarker := FALSE;
//	ELSIF MyLaser1.P_bError THEN
//		bDisconnectFromLaserMarker := FALSE;
//		MyLaser1.M_ClearError();
//	END_IF
//END_IF


//IF bPeakCurrentProgramInLaser THEN
//	bRes_PeakCurrentProgramInLaser := MyLaser1.M_PeakCurrentProgram();
//	IF bRes_PeakCurrentProgramInLaser THEN
//		bPeakCurrentProgramInLaser := FALSE;
//	ELSIF MyLaser1.P_bError THEN
//		bPeakCurrentProgramInLaser := FALSE;
//		MyLaser1.M_ClearError();
//	END_IF
//END_IF


//IF bSendProgramToLaser THEN
//	bRes_SendProgramtoLaser := MyLaser1.M_SendProgramtoLaser(filepath,LaserMemoryLocation);
//	IF bRes_SendProgramtoLaser THEN
//		bSendProgramToLaser := FALSE;
//	ELSIF MyLaser1.P_bError THEN
//		bSendProgramToLaser := FALSE;
//		MyLaser1.M_ClearError();
//	END_IF
//END_IF

//IF bSaveCurrentLaserProgramtoPC THEN
//	bRes_SaveCurrentLaserProgramtoPC := MyLaser1.M_SaveCurrentLaserProgramtoPC(LaserProgramFolderPath, out_bool_SaveProgramToPC_Success => SaveCurrentLaserProgramToPCSuccess);
//	IF bRes_SaveCurrentLaserProgramtoPC THEN
////		SaveCurrentLaserProgramToPCSuccess := MyLaser1
//		bSaveCurrentLaserProgramtoPC := FALSE;
//	ELSIF MyLaser1.P_bError THEN
//		bSaveCurrentLaserProgramtoPC := FALSE;
//		MyLaser1.M_ClearError();
//	END_IF
//END_IF

//IF bGetCurrentProgram THEN
//	bRes_GetCurrentProgram := MyLaser1.M_GetCurrentProgram(strCurrentProgram => CurrentProgramName);
//	IF bRes_GetCurrentProgram THEN
//		bGetCurrentProgram := FALSE;
//	ELSIF MyLaser1.P_bError THEN
//		bGetCurrentProgram := FALSE;
//		MyLaser1.M_ClearError();
//	END_IF
//END_IF

//IF bStartMarking THEN
//	bRes_StartMarking := MyLaser1.M_StartMarking();
//	IF bRes_StartMarking THEN
//		bStartMarking := FALSE;
//	ELSIF MyLaser1.P_bError THEN
//		bStartMarking := FALSE;
//		MyLaser1.M_ClearError();
//	END_IF
//END_IF

//IF bStopMarking THEN
//	bRes_StopMarking := MyLaser1.M_StopMarking();
//	IF bRes_StopMarking THEN
//		bStopMarking := FALSE;
//	ELSIF MyLaser1.P_bError THEN
//		bStopMarking := FALSE;
//		MyLaser1.M_ClearError();
//	END_IF
//END_IF

//IF bResetErrors THEN
//	bRes_Reset := MyLaser1.M_Reset();
//	IF bRes_Reset THEN
//		bResetErrors := FALSE;
//	ELSIF MyLaser1.P_bError THEN
//		bResetErrors := FALSE;
//		MyLaser1.M_ClearError();
//	END_IF
//END_IF

////IF bUpdateProgramBlockInTheLaser THEN
////	bRes_UpdateProgramBlockInTheLaser := MyLaser1.M_UpdateSingleProgramBlockData(LaserMemoryLocation, _blockNumber, _blockData, _blockType, out_bool_UpdateData_Success => _bUpdateSingleBlockDataSuccess);
////	IF bRes_UpdateProgramBlockInTheLaser THEN
////		bUpdateProgramBlockInTheLaser := FALSE;
////	ELSIF MyLaser1.P_bError THEN
////		bUpdateProgramBlockInTheLaser := FALSE;
////		MyLaser1.M_ClearError();
////	END_IF
////END_IF

//IF bUpdateProgramBlockInTheLaser THEN
//	bRes_UpdateProgramBlockInTheLaser := MyLaser1.M_UpdateSingleBlockMarkingInformation(_blockNumber, _blockData, _bool_markenabled);
//	IF bRes_UpdateProgramBlockInTheLaser THEN
//		bUpdateProgramBlockInTheLaser := FALSE;
//	ELSIF MyLaser1.P_bError THEN
//		bUpdateProgramBlockInTheLaser := FALSE;
//		MyLaser1.M_ClearError();
//	END_IF
//END_IF

//IF bUpdateProgramBlockMarkEnabledInTheLaser THEN
//	bRes_UpdateProgramBlockMarkEnabledInTheLaser := MyLaser1.M_UpdateSingleProgramBlockMarkEnabled( LaserProgramMemoryLocation := LaserMemoryLocation, BlockNumber := _blockNumber, BlockType := _blockType ,MarkEnabled := _bool_markenabled ,out_bool_MarkEnabled_Success => _bUpdateSingleBlockMarkEnabled_Success);
//	IF bRes_UpdateProgramBlockMarkEnabledInTheLaser THEN
//		bUpdateProgramBlockMarkEnabledInTheLaser := FALSE;
//	ELSIF MyLaser1.P_bError THEN
//		bUpdateProgramBlockMarkEnabledInTheLaser := FALSE;
//		MyLaser1.M_ClearError();
//	END_IF
//END_IF

//IF bGetLaserStatus THEN
//	bRes_GetLaserStatus := MyLaser1.M_GetLaserStatus( out_string_laserStatus => _string_laserstatus);
//	IF bRes_GetLaserStatus THEN
//		bGetLaserStatus := FALSE;
//	ELSIF MyLaser1.P_bError THEN
//		bGetLaserStatus := FALSE;
//		MyLaser1.M_ClearError();
//	END_IF
//END_IF

//IF bGetLaserErrorStatus THEN
//	bRes_GetLaserErrorStatus := MyLaser1.M_GetLaserErrorStatus( out_bool_IsLaserError => _bIsLaserError);
//	IF bRes_GetLaserErrorStatus THEN
//		bGetLaserErrorStatus := FALSE;
//	ELSIF MyLaser1.P_bError THEN
//		bGetLaserErrorStatus := FALSE;
//		MyLaser1.M_ClearError();
//	END_IF
//END_IF

//IF bGetLaserActivatedStatus THEN
//	bRes_GetLaserActivatedStatus := MyLaser1.M_GetLaserActivatedStatus( out_IsLaserActivated => _bIsLaserActivated);
//	IF bRes_GetLaserActivatedStatus THEN
//		bGetLaserActivatedStatus := FALSE;
//	ELSIF MyLaser1.P_bError THEN
//		bGetLaserActivatedStatus := FALSE;
//		MyLaser1.M_ClearError();
//	END_IF
//END_IF

//IF bGetLaserMarkingStatus THEN
//	bRes_GetLaserMarkingStatus := MyLaser1.M_GetLaserMarkingStatus( out_bool_IsLaserMarking => _bIsLaserMarking);
//	IF bRes_GetLaserMarkingStatus THEN
//		bGetLaserMarkingStatus := FALSE;
//	ELSIF MyLaser1.P_bError THEN
//		bGetLaserMarkingStatus := FALSE;
//		MyLaser1.M_ClearError();
//	END_IF
//END_IF

//IF _OneTimeArrayBuild THEN
//	FOR intIndex2 := 0 TO 255 DO
//		IF intIndex2 <= LastBlockToMark THEN
//			BlockInfoArray[intIndex2].MarkEnabled := TRUE;
//			_tempString := CONCAT('Block', INT_TO_STRING(intIndex2));
//			BlockInfoArray[intIndex2].BlockText := _tempString;
//		ELSE
//			BlockInfoArray[intIndex2].MarkEnabled := FALSE;	
//			BlockInfoArray[intIndex2].BlockText := '';
//		END_IF
//	END_FOR
//	_OneTimeArrayBuild := FALSE;
//END_IF

//IF bUpdateAllMarkingInfo_MethodCall THEN
//	bRes_UpdateAllMarkingInfo_MethodCall := MyLaser1.M_UpdateAllMarkingInformation(LastBlockToMark);
//	bUpdateAllMarkingInfo_MethodCall := FALSE;
//END_IF
//IF MyLaser1.P_bError THEN
//	bUpdateAllMarkingInfo_MethodCall := FALSE;
//	MyLaser1.M_ClearError();
//END_IF

//IF bUpdateAllMarkingInfo THEN
//	CASE inst_intStep OF
//		0: //Check for errors and Integer value which we are gonna run the update single block information
//				IF MyLaser1.P_bError THEN
//					inst_intStep := 0;
//					bUpdateAllMarkingInfo := FALSE;
//				ELSE
//					inst_intStep := 10;
//				END_IF
//		10: // Run the M_UpdateSingleBlockMarkingInformation Command
//				bRes_UpdateAllMarkInfo[intIndex] := MyLaser1.M_UpdateSingleBlockMarkingInformation(intIndex ,BlockInfoArray[intIndex].BlockText, BlockInfoArray[intIndex].MarkEnabled);
//				IF bRes_UpdateAllMarkInfo[intIndex] THEN 
//					inst_intStep := 20;
//				ELSIF MyLaser1.P_bError THEN
//					inst_intStep := 0;
//					intIndex :=0;
//					bUpdateAllMarkingInfo := FALSE;
//				END_IF
//		20: // Check if the M_UpdateSingleBlockMarkingInformation command failed or passed
//				IF bRes_UpdateAllMarkInfo[LastBlockToMark] OR NOT bRes_UpdateAllMarkInfo[intIndex] OR (intIndex = LastBlockToMark) THEN //This means we reached the final element update
//					bUpdateAllMarkingInfo := FALSE;
//					intIndex :=0;
//					inst_intStep := 0;
//				ELSIF bRes_UpdateAllMarkInfo[intIndex] THEN
//					inst_intStep := 0;
//					intIndex := intIndex + 1;
//				ELSIF MyLaser1.P_bError THEN
//					bUpdateAllMarkingInfo := FALSE;
//					MyLaser1.M_ClearError();	
//				END_IF			
//	END_CASE
//END_IF

//IF bGetLimitsFromDB THEN
//	_inst_bDataTransferred := fbDataHandler.M_TransferData(in_strParametersDatabaseName);
//	IF _inst_bDataTransferred THEN
//		bGetLimitsFromDB := FALSE;
//	ELSIF fbDataHandler.P_bError THEN
//		bGetLimitsFromDB := FALSE;
//		fbDataHandler.M_ClearError();
//	END_IF
//END_IF

//IF bGetLaserParamsFromDB_L1 THEN
//	_inst_bLaserLimitsDataTransferred_L1 := fbDataHandler.M_TransferData(in_strParametersDBNameLaserLimits_L1);
//	IF _inst_bLaserLimitsDataTransferred_L1 THEN
//		bGetLaserParamsFromDB_L1 := FALSE;
//		ELSIF fbDataHandler.P_bError THEN
//			bGetLaserParamsFromDB_L1 := FALSE;
//			fbDataHandler.M_ClearError();
//	END_IF
//END_IF

//IF bGetLaserParamsFromDB_L2 THEN
//	_inst_bLaserLimitsDataTransferred_L2 := fbDataHandler.M_TransferData(in_strParametersDBNameLaserLimits_L2);
//	IF _inst_bLaserLimitsDataTransferred_L2 THEN
//		bGetLaserParamsFromDB_L2 := FALSE;
//		ELSIF fbDataHandler.P_bError THEN
//			bGetLaserParamsFromDB_L2 := FALSE;
//			fbDataHandler.M_ClearError();
//	END_IF
//END_IF

//IF bGetLaserParamsFromDB_R1 THEN
//	_inst_bLaserLimitsDataTransferred_R1 := fbDataHandler.M_TransferData(in_strParametersDBNameLaserLimits_R1);
//	IF _inst_bLaserLimitsDataTransferred_R1 THEN
//		bGetLaserParamsFromDB_R1 := FALSE;
//		ELSIF fbDataHandler.P_bError THEN
//			bGetLaserParamsFromDB_R1 := FALSE;
//			fbDataHandler.M_ClearError();
//	END_IF
//END_IF

//IF bGetLaserParamsFromDB_R2 THEN
//	_inst_bLaserLimitsDataTransferred_R2 := fbDataHandler.M_TransferData(in_strParametersDBNameLaserLimits_R2);
//	IF _inst_bLaserLimitsDataTransferred_R2 THEN
//		bGetLaserParamsFromDB_R2 := FALSE;
//		ELSIF fbDataHandler.P_bError THEN
//			bGetLaserParamsFromDB_R2 := FALSE;
//			fbDataHandler.M_ClearError();
//	END_IF
//END_IF

//IF bPerformPriorOp_Smart THEN
//	_inst_bPriorOp_Smart := fbDataHandler2.M_TransferData(in_strParametersDBName_SmartWater);
//	IF _inst_bPriorOp_Smart THEN
//		bPerformPriorOp_Smart := FALSE;
//	ELSIF fbDataHandler2.P_bError THEN 
//		bPerformPriorOp_Smart := FALSE;
//		fbDataHandler2.M_ClearError();
//	END_IF
//END_IF

//IF bPerformPriorOp_FFT THEN
//	_inst_bPriorOp_FFT := fbDataHandler.M_TransferData(in_strParametersDBName_FFTLaser_L1);
//	IF _inst_bPriorOp_FFT THEN
//		bPerformPriorOp_FFT := FALSE;
//	ELSIF fbDataHandler.P_bError THEN 
//		bPerformPriorOp_FFT := FALSE;
//		fbDataHandler.M_ClearError();
//	END_IF
//END_IF

//Temp_CR_LOOKUP_NestL1 := FIND('GV354-006:220705-141019_CR','_CR');
//iLengthDataMatrixNestL1 := LEN('GV354-006:220705-141019_CR');
//IF  (Temp_CR_LOOKUP_NestL1 > 0) THEN
//	ParamsArrayNestA := REPLACE('GV354-006:220705-141019_CR', concat(' CR ' , '0.023456'),6,iLengthDataMatrixNestL1 - 2);
//END_IF
END_METHOD

METHOD M_TestMESVars : BOOL
VAR_INPUT
	
END_VAR
VAR
	//MES Data Tracking Testing
//	fbDataHandler3: FB_MESDataTracking;
//	bPerformGetLotInfoFromLotBarcode: BOOL;
//	_inst_bGetLotInfo_LotBarcode: BOOL;
//	in_strParamDBName_GetLotInfo: T_MaxString := 'GetLotInfo1';
	
//	bPerformGetOpInfoFromOpBarcode: BOOL;
//	in_strParamDBName_GetOpInfo: T_MaxString := 'GetOperatorInfo1';
//	_inst_bGetOpInfo_OpBarcode: BOOL;
	
//	bPerformStartLot : BOOL;
//	_inst_bStartLot : BOOL;
//	in_strParamDBName_StartLot : T_MaxString := 'StartLot1';
	
//	bPerformGetProdLotComponents : BOOL;
//	_inst_bGetProdLotComponents : BOOL;
//	in_strParamDBName_GetProdLotComps : T_MaxString := 'GetProdLotComponents1';
	
//	bPerformComponentValidation1 : BOOL;
//	_inst_bCompValidation1 : BOOL;
//	in_strParamDBName_Comp1Validation1 : T_MaxString := 'ComponentValidation1';
	
//	bPerformComponentValidation2 : BOOL;
//	_inst_bCompValidation2 : BOOL;
//	in_strParamDBName_Comp1Validation2 : T_MaxString := 'ComponentValidation2';
	
//	bPerformComponentValidation3 : BOOL;
//	_inst_bCompValidation3 : BOOL;
//	in_strParamDBName_Comp1Validation3 : T_MaxString := 'ComponentValidation3';
	
//	bPerformGetMachineSettings : BOOL;
//	_inst_bGetMachineSettings : BOOL;
//	in_strParamDBName_GetMachSetting : T_MaxString := 'GetMachineSettings1';
	
//	bPerformAddScrapCompByReason : BOOL;
//	_inst_bAddScrapCompByReason : BOOL;
//	in_strParamDBName_AddScrapCompByReason : T_MaxString := 'AddScrapComponentByReason1';
	
//	bPerformEndLotComp : BOOL;
//	_inst_bEndLotComp : BOOL;
//	in_strParamDBName_EndLotComp : T_MaxString := 'EndLotComponent1';
	
//	bPerformGetMachineDefects : BOOL;
//	_inst_bGetMachineDefects : BOOL;
//	in_strParamDBName_GetMachDefects : T_MaxString := 'GetMachineDefects1';
END_VAR

//IF bPerformGetLotInfoFromLotBarcode THEN
//	_inst_bGetLotInfo_LotBarcode := fbDataHandler3.M_TransferData(in_strParamDBName_GetLotInfo);
//	IF _inst_bGetLotInfo_LotBarcode THEN
//		bPerformGetLotInfoFromLotBarcode := FALSE;
//	ELSIF fbDataHandler3.P_bError THEN 
//		bPerformGetLotInfoFromLotBarcode := FALSE;
//		fbDataHandler3.M_ClearError();
//	END_IF
//END_IF

//IF bPerformGetOpInfoFromOpBarcode THEN
//	_inst_bGetOpInfo_OpBarcode := fbDataHandler3.M_TransferData(in_strParamDBName_GetOpInfo);
//	IF _inst_bGetOpInfo_OpBarcode THEN
//		bPerformGetOpInfoFromOpBarcode := FALSE;
//	ELSIF fbDataHandler3.P_bError THEN 
//		bPerformGetOpInfoFromOpBarcode := FALSE;
//		fbDataHandler3.M_ClearError();
//	END_IF
//END_IF

//IF bPerformStartLot THEN
//	_inst_bStartLot := fbDataHandler3.M_TransferData(in_strParamDBName_StartLot);
//	IF _inst_bStartLot THEN
//		bPerformStartLot := FALSE;
//	ELSIF fbDataHandler3.P_bError THEN 
//		bPerformStartLot := FALSE;
//		fbDataHandler3.M_ClearError();
//	END_IF
//END_IF

//IF bPerformGetProdLotComponents THEN
//	_inst_bGetProdLotComponents := fbDataHandler3.M_TransferData(in_strParamDBName_GetProdLotComps);
//	IF _inst_bGetProdLotComponents THEN
//		bPerformGetProdLotComponents := FALSE;
//	ELSIF fbDataHandler3.P_bError THEN 
//		bPerformGetProdLotComponents := FALSE;
//		fbDataHandler3.M_ClearError();
//	END_IF
//END_IF


//IF bPerformComponentValidation1 THEN
//	_inst_bCompValidation1 := fbDataHandler3.M_TransferData(in_strParamDBName_Comp1Validation1);
//	IF _inst_bCompValidation1 THEN
//		bPerformComponentValidation1 := FALSE;
//	ELSIF fbDataHandler3.P_bError THEN 
//		bPerformComponentValidation1 := FALSE;
//		fbDataHandler3.M_ClearError();
//	END_IF
//END_IF

//IF bPerformComponentValidation2 THEN
//	_inst_bCompValidation2 := fbDataHandler3.M_TransferData(in_strParamDBName_Comp1Validation2);
//	IF _inst_bCompValidation2 THEN
//		bPerformComponentValidation2 := FALSE;
//	ELSIF fbDataHandler3.P_bError THEN 
//		bPerformComponentValidation2 := FALSE;
//		fbDataHandler3.M_ClearError();
//	END_IF
//END_IF

//IF bPerformComponentValidation3 THEN
//	_inst_bCompValidation3 := fbDataHandler3.M_TransferData(in_strParamDBName_Comp1Validation3);
//	IF _inst_bCompValidation3 THEN
//		bPerformComponentValidation3 := FALSE;
//	ELSIF fbDataHandler3.P_bError THEN 
//		bPerformComponentValidation3 := FALSE;
//		fbDataHandler3.M_ClearError();
//	END_IF
//END_IF

//IF bPerformGetMachineSettings THEN
//	_inst_bGetMachineSettings := fbDataHandler3.M_TransferData(in_strParamDBName_GetMachSetting);
//	IF _inst_bGetMachineSettings THEN
//		bPerformGetMachineSettings := FALSE;
//	ELSIF fbDataHandler3.P_bError THEN 
//		bPerformGetMachineSettings := FALSE;
//		fbDataHandler3.M_ClearError();
//	END_IF
//END_IF

//IF bPerformAddScrapCompByReason THEN
//	_inst_bAddScrapCompByReason := fbDataHandler3.M_TransferData(in_strParamDBName_AddScrapCompByReason);
//	IF _inst_bAddScrapCompByReason THEN
//		bPerformAddScrapCompByReason := FALSE;
//	ELSIF fbDataHandler3.P_bError THEN 
//		bPerformAddScrapCompByReason := FALSE;
//		fbDataHandler3.M_ClearError();
//	END_IF
//END_IF

//IF bPerformEndLotComp THEN
//	_inst_bEndLotComp := fbDataHandler3.M_TransferData(in_strParamDBName_EndLotComp);
//	IF _inst_bEndLotComp THEN
//		bPerformEndLotComp := FALSE;
//	ELSIF fbDataHandler3.P_bError THEN 
//		bPerformEndLotComp := FALSE;
//		fbDataHandler3.M_ClearError();
//	END_IF
//END_IF

//IF bPerformGetMachineDefects THEN
//	_inst_bGetMachineDefects := fbDataHandler3.M_TransferData(in_strParamDBName_GetMachDefects);
//	IF _inst_bGetMachineDefects THEN
//		bPerformGetMachineDefects := FALSE;
//	ELSIF fbDataHandler3.P_bError THEN 
//		bPerformGetMachineDefects := FALSE;
//		fbDataHandler3.M_ClearError();
//	END_IF
//END_IF
END_METHOD

END_PROGRAM

// ---- 1 Module/0 Machines/FB_ExampleMachine.TcPOU
FUNCTION_BLOCK FB_ExampleMachine EXTENDS FB_Machine IMPLEMENTS I_SimpleStateful
VAR_INPUT
	in_fbStation1: REFERENCE TO FB_Station;
	in_fbStation2: REFERENCE TO FB_Station;
	in_fbStation3: REFERENCE TO FB_Station;
	in_fbStation4: REFERENCE TO FB_Station;
	
	in_bAbortBtn: BOOL;
	in_bResetBtn: BOOL;
	in_bStartBtn: BOOL;
	in_bStopBtn: BOOL;
	in_bSuspendBtn: BOOL;
END_VAR
VAR_OUTPUT
END_VAR
VAR
END_VAR

THIS^.M_SetStation(1, in_fbStation1);
THIS^.M_SetStation(2, in_fbStation2);
THIS^.M_SetStation(3, in_fbStation3);
THIS^.M_SetStation(4, in_fbStation4);

THIS^.A_StateMachine();

(* The 'Aborting' state can be entered at any time while within the 'abortable'
section of the state machine. It is typically entered in response to an 'Abort'
command or a critical fault. The logic should safely but rapidly bring the
components of the module to a stop while maintaining as much information about
the pre-abort scenario as possible. *)
METHOD M001_Aborting : BOOL
VAR_OUTPUT
	(* This should be set to true once all components of the module have safely
	come to a stop. Once set to true, the state machine will move to the
	'Aborted' state. *)
	bAborted	: BOOL;
END_VAR
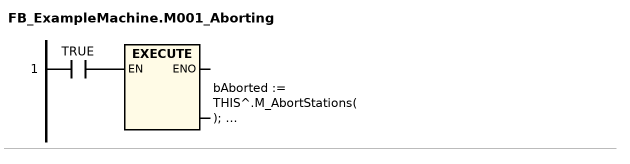
// NETWORK 1
bAborted := THIS^.M_AbortStations();
END_METHOD

(* This state is entered after the aborting state completes, and should
not modify anything in the module while awaiting an explicit 'Clear' command. *)
METHOD M011_Aborted : BOOL
VAR_OUTPUT
	(* This should be set to true once an explicit 'Clear' command is received.
	Once set to true, the state machine will move to the 'Clearing' state. *)
	bClear	: BOOL;
END_VAR
VAR_INST // added by the converter: edge detectors and wires of the graphical bodies
    _rt1 : R_TRIG;
END_VAR
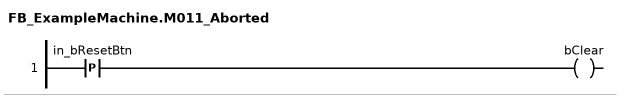
// NETWORK 1
_rt1(CLK := in_bResetBtn);
bClear := _rt1.Q;
END_METHOD

(* This state should clear any faults and reset any safety features related
to the module, as well as perform actions similar to the 'Stopping' state
if they were not already performed while aborting. *)
METHOD M021_Clearing : BOOL
VAR_OUTPUT
	(* This should be set to true once the safety state of all module
	components are reset and all errors are cleared. *)
	bCleared	: BOOL;
	(* This should be set to true if a potentially hazardous error or a safety
	fault has occurred in any tasks. Once set to true, the state machine will
	move to the 'Aborting' state. *)
	bAbort	: BOOL;
END_VAR
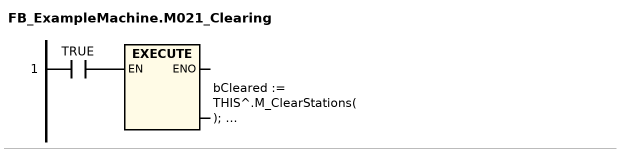
// NETWORK 1
bCleared := THIS^.M_ClearStations();
END_METHOD

(* This state can be entered from anywhere within the 'stoppable' group of
states. This state should safely bring the components of the module to a
controlled stop and then move to the 'Stopped' state once completed. *)
METHOD M101_Stopping : BOOL
VAR_OUTPUT
	(* This should be set to true once all relevant components have come to a
	controlled stop. Once set to true, the state machine will move to the
	'Stopped' state. *)
	bStopped	: BOOL;
	(* This should be set to true if a potentially hazardous error or a safety
	fault has occurred in any tasks. Once set to true, the state machine will
	move to the 'Aborting' state. *)
	bAbort	: BOOL;
END_VAR
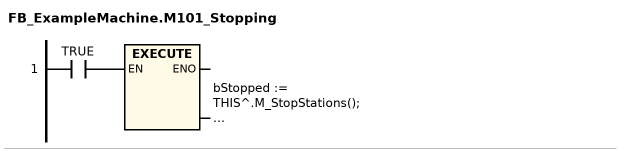
// NETWORK 1
bStopped := THIS^.M_StopStations();
END_METHOD

(* The machine should be stationary and awaiting an explicit 'Reset' command
while in this state. Once the 'Reset' command is received, the state machine
will move to the 'Resetting' state. *)
METHOD M111_Stopped : BOOL
VAR_OUTPUT
	(* This should be set to true if an explicit reset command is received.
	Once set to true, the state machine will move to the 'Resetting' state. *)
	bReset	: BOOL;
	(* This should be set to true if a potentially hazardous error or a safety
	fault has occurred in any tasks. Once set to true, the state machine will
	move to the 'Aborting' state. *)
	bAbort	: BOOL;
END_VAR
VAR_INST // added by the converter: edge detectors and wires of the graphical bodies
    _rt1 : R_TRIG;
END_VAR
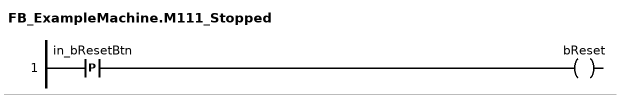
// NETWORK 1
_rt1(CLK := in_bResetBtn);
bReset := _rt1.Q;
END_METHOD

(* This state should place the module and all of its components into a safe
energized idle state where it will wait for a start command. Once all tasks are
complete, it will move to the 'Idle' state. No external movement should occur
as a result of this state. *)
METHOD M201_Resetting : BOOL
VAR_OUTPUT
	(* Set this to true once the module is energized and ready to start.
	Once set to true, the state machine will move to the 'Idle' state. *)
	bIdle	: BOOL;
	(* This should be set to true if an external source requests that the module
	exit its current state and come to a controlled stop. Once set to true, the
	state machine will move to the 'Stopping' state. *)
	bStop	: BOOL;
	(* This should be set to true if a potentially hazardous error or a safety
	fault has occurred in any tasks. Once set to true, the state machine will
	move to the 'Aborting' state. *)
	bAbort	: BOOL;
END_VAR
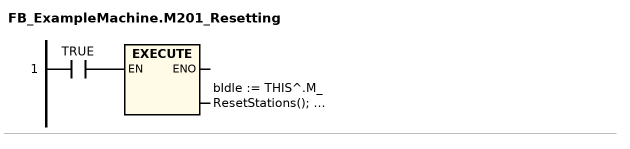
// NETWORK 1
bIdle := THIS^.M_ResetStations();
END_METHOD

(* This state should maintain the status of the module and its components that
was set by the resetting step while awaiting an explicit 'Start' command. *)
METHOD M211_Idle : BOOL
VAR_OUTPUT
	(* This should be set to true if an explicit 'Start' command is received.
	Once set to true, the state machine will move to the 'Starting' state. *)
	bStart	: BOOL;
	(* This should be set to true if an external source requests that the module
	exit its current state and come to a controlled stop. Once set to true, the
	state machine will move to the 'Stopping' state. *)
	bStop	: BOOL;
	(* This should be set to true if a potentially hazardous error or a safety
	fault has occurred in any tasks. Once set to true, the state machine will
	move to the 'Aborting' state. *)
	bAbort	: BOOL;
END_VAR
VAR_INST // added by the converter: edge detectors and wires of the graphical bodies
    _rt1 : R_TRIG;
END_VAR
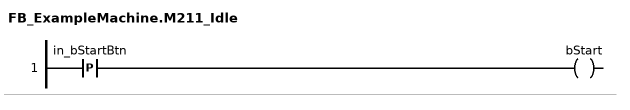
// NETWORK 1
_rt1(CLK := in_bStartBtn);
bStart := _rt1.Q;
END_METHOD

(* This state should make any final preparations needed for the 'Execute' state
prior to entering the 'Execute' state. *)
METHOD M301_Starting : BOOL
VAR_OUTPUT
	(* This should be set to true once the module and its components are fully
	prepared for process execution. Once set to true, the state machine will
	move to the 'Execute' state. *)
	bStarted	: BOOL;
	(* This should be set to true if an external source requests that the module
	exit its current state and come to a controlled stop. Once set to true, the
	state machine will move to the 'Stopping' state. *)
	bStop	: BOOL;
	(* This should be set to true if a potentially hazardous error or a safety
	fault has occurred in any tasks. Once set to true, the state machine will
	move to the 'Aborting' state. *)
	bAbort	: BOOL;
END_VAR
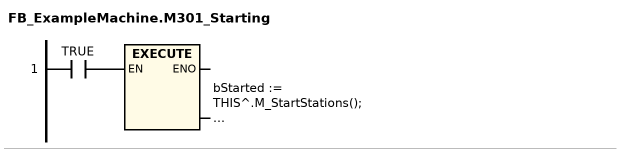
// NETWORK 1
bStarted := THIS^.M_StartStations();
END_METHOD

(* The module should remain in this state while it is actively performing
automated tasks. Once all work is finished the state machine should move to the
'Completing' state. *)
METHOD M311_Execute : BOOL
VAR_OUTPUT
	(* This should be set to true once all tasks are complete and automated
	execution should be ended. Once set to true, the state machine will move to
	the 'Completing' state. *)
	bFinished	: BOOL;
	(* This should be set to true as a result of an explicit 'Hold' command
	or if internal conditions require the module to stop operation without
	completely exiting the execution sequence. Once set to true, the state
	machine will move to the 'Holding' state. *)
	bHold	: BOOL;
	(* This should be set to true if external conditions require the module to
	suspend operation until the external conditions are cleared. Once set to
	true, the state machine will move to the 'Suspending' state. *)
	bSuspend	: BOOL;
	(* This should be set to true if an external source requests that the module
	exit its current state and come to a controlled stop. Once set to true, the
	state machine will move to the 'Stopping' state. *)
	bStop	: BOOL;
	(* This should be set to true if a potentially hazardous error or a safety
	fault has occurred in any tasks. Once set to true, the state machine will
	move to the 'Aborting' state. *)
	bAbort	: BOOL;
END_VAR
VAR_INST // added by the converter: edge detectors and wires of the graphical bodies
    _rt1 : R_TRIG;
END_VAR
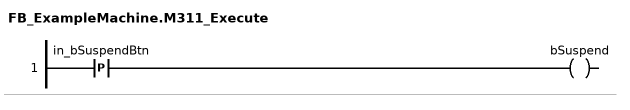
// NETWORK 1
_rt1(CLK := in_bSuspendBtn);
bSuspend := _rt1.Q;
END_METHOD

(* This state will perform any post-execution tasks prior to moving to the
'Completed' state. *)
METHOD M321_Completing : BOOL
VAR_OUTPUT
	(* Move to the Complete state*)
	bCompleted	: BOOL;
	(* This should be set to true if an external source requests that the module
	exit its current state and come to a controlled stop. Once set to true, the
	state machine will move to the 'Stopping' state. *)
	bStop	: BOOL;
	(* This should be set to true if a potentially hazardous error or a safety
	fault has occurred in any tasks. Once set to true, the state machine will
	move to the 'Aborting' state. *)
	bAbort	: BOOL;
END_VAR
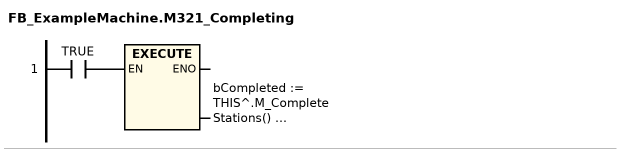
// NETWORK 1
bCompleted := THIS^.M_CompleteStations();
END_METHOD

(* The module should remain stationary within this state while maintaing any
execution statistics and awaiting an explicit 'Return' command. *)
METHOD M331_Complete : BOOL
VAR_OUTPUT
	(* This should be set to true if an explicit 'Return' command is received.
	Once set to true, the state machine will move to the 'Resetting' state. *)
	bReturn	: BOOL;
	(* This should be set to true if an external source requests that the module
	exit its current state and come to a controlled stop. Once set to true, the
	state machine will move to the 'Stopping' state. *)
	bStop	: BOOL;
	(* This should be set to true if a potentially hazardous error or a safety
	fault has occurred in any tasks. Once set to true, the state machine will
	move to the 'Aborting' state. *)
	bAbort	: BOOL;
END_VAR
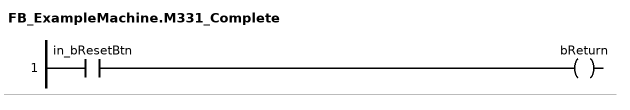
// NETWORK 1
bReturn := in_bResetBtn;
END_METHOD

(* This state should safely pause task executions without completely ending or
resetting them. *)
METHOD M401_Holding : BOOL
VAR_OUTPUT
	(* This should be set to true once all execution tasks are safely paused.
	Once set to true, the state machine will move to the 'Held' state. *)
	bHeld	: BOOL;
	(* This should be set to true if an external source requests that the module
	exit its current state and come to a controlled stop. Once set to true, the
	state machine will move to the 'Stopping' state. *)
	bStop	: BOOL;
	(* This should be set to true if a potentially hazardous error or a safety
	fault has occurred in any tasks. Once set to true, the state machine will
	move to the 'Aborting' state. *)
	bAbort	: BOOL;
END_VAR
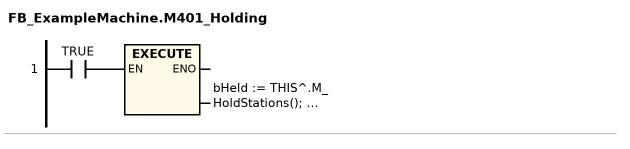
// NETWORK 1
bHeld := THIS^.M_HoldStations();
END_METHOD

(* In this state the most recent execution status should be maintained while
awaiting an explicit 'Unhold' command once internal conditions are satisfactory. *)
METHOD M411_Held : BOOL
VAR_OUTPUT
	(* This should be set to true if an explicit 'Unhold' command is received.
	Once set to true, the state machine will move to the 'Unholding' state. *)
	bUnhold	: BOOL;
	(* This should be set to true if an external source requests that the module
	exit its current state and come to a controlled stop. Once set to true, the
	state machine will move to the 'Stopping' state. *)
	bStop	: BOOL;
	(* This should be set to true if a potentially hazardous error or a safety
	fault has occurred in any tasks. Once set to true, the state machine will
	move to the 'Aborting' state. *)
	bAbort	: BOOL;
END_VAR
VAR_INST // added by the converter: edge detectors and wires of the graphical bodies
    _rt1 : R_TRIG;
END_VAR
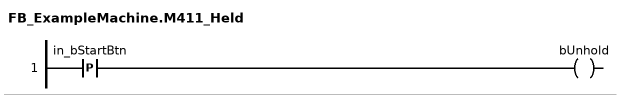
// NETWORK 1
_rt1(CLK := in_bStartBtn);
bUnhold := _rt1.Q;
END_METHOD

(* In this state, the module and its components should be returned to the
scenario it was in before it entered the 'Holding' step so that the
'Execute' state can pick up where it left off. *)
METHOD M421_Unholding : BOOL
VAR_OUTPUT
	(* This should be set to true once the module is ready to restart
	execution. Once set to true, the state machine will move to the 'Execute'
	state. *)
	bUnheld	: BOOL;
	(* This should be set to true if an external source requests that the module
	exit its current state and come to a controlled stop. Once set to true, the
	state machine will move to the 'Stopping' state. *)
	bStop	: BOOL;
	(* This should be set to true if a potentially hazardous error or a safety
	fault has occurred in any tasks. Once set to true, the state machine will
	move to the 'Aborting' state. *)
	bAbort	: BOOL;
END_VAR
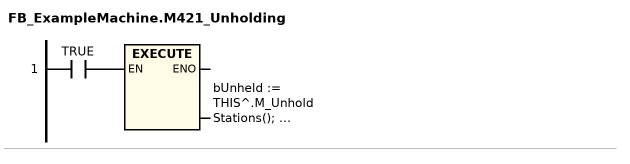
// NETWORK 1
bUnheld := THIS^.M_UnholdStations();
END_METHOD

(* This state should safely pause task executions without completely ending or
resetting them. *)
METHOD M501_Suspending : BOOL
VAR_OUTPUT
	(* This should be set to true once all execution tasks are safely paused.
	Once set to true, the state machine will move to the 'Suspended' state. *)
	bSuspended	: BOOL;
	(* This should be set to true if an external source requests that the module
	exit its current state and come to a controlled stop. Once set to true, the
	state machine will move to the 'Stopping' state. *)
	bStop	: BOOL;
	(* This should be set to true if a potentially hazardous error or a safety
	fault has occurred in any tasks. Once set to true, the state machine will
	move to the 'Aborting' state. *)
	bAbort	: BOOL;
END_VAR
